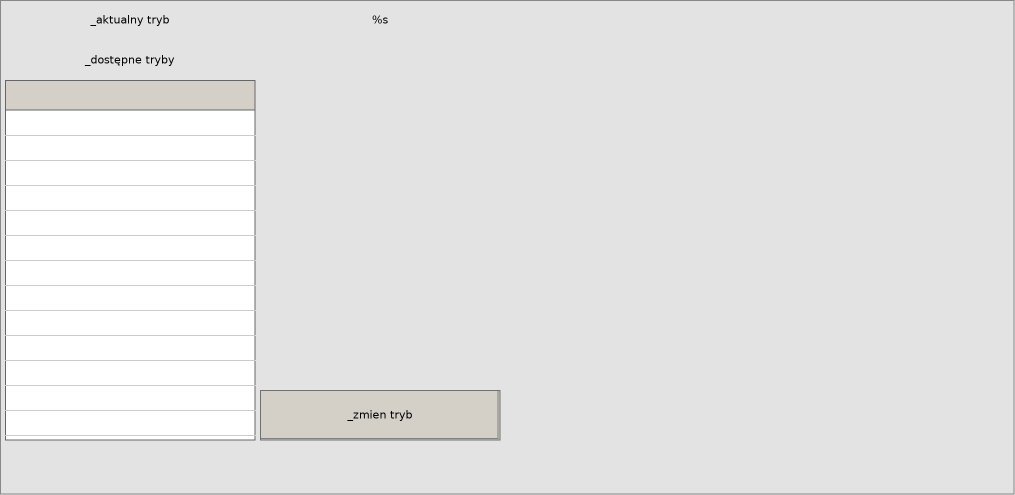
VISUALIZATION F_04_ChangeMode  // 1015x495
VAR_IN_OUT
	stScreenData	: ST_MCHMIPrepareScreen_04_XX;
	
END_VAR
    Rectangle (5,45 250x30), "_dostępne tryby", text list: 'TextList_04', text index: 0
    Table (5,80 250x360), data array: stScreenData.arrNamesOfMode
        p3854506369: stScreenData.arrNamesOfMode[INDEX].wsDescription
        p1892666644: stScreenData.arrNamesOfMode[INDEX].iNumber
        p1128707560: stScreenData.iNumberModeToDisplay-1
        p1137915858: stScreenData.iSelectedMode
        p1822360349: stScreenData.bSelectedRow
    Rectangle (5,5 250x30), "_aktualny tryb", text list: 'TextListGlobal', text index: 1
    Rectangle (255,5 250x30), "%s", text variable: stScreenData.wsActualMode
    Button (260,390 240x50), "_zmien tryb", text list: 'TextList_04', text index: 1
        OnMouseDown: execute { stScreenData.bChangeMode := TRUE; }
END_VISUALIZATION

(* stored: Version 1.1.0.1
   Visu F_04_ChangeMode: Id {0b9f0e63-371a-0c07-24bf-de3c4cd40d7e} *)
